// List of Strings.
FUNCTION_BLOCK FB_StringList
VAR
   List : ARRAY[0..GVL_List.LIST_SIZE - 1] OF T_MaxString; // hold list
   _Count : UDINT := 0; // number of items.
END_VAR

// Add item to list. TRUE if successful. 
METHOD PUBLIC AddItem : BOOL
VAR_INPUT
   Item : T_MaxString; // item to add.
END_VAR
IF _Count < GVL_List.LIST_SIZE THEN
   List[_Count] := Item; // list is zero indexed, so number of items points at next free space.
   _Count := _Count + 1;
   AddItem := TRUE;
END_IF
END_METHOD

// Removes all list items
METHOD PUBLIC Clear
MEMSET(ADR(List[0]), 0, SIZEOF(List));
_Count := 0;
END_METHOD

// TRUE if Item is in FB_List.
METHOD PUBLIC Contains : BOOL
VAR_INPUT
   Item : T_MaxString; // Item to check.
END_VAR
Contains := FindIndex(Item) >= 0;
END_METHOD

// TRUE if supplied key part is in any entry
METHOD PUBLIC ContainsPartial : BOOL
VAR_INPUT
   PartialItem : T_MaxString;
END_VAR
ContainsPartial := FindIndexPartialKey(PartialItem) >= 0;
END_METHOD

METHOD CopyList
VAR_IN_OUT
   ListToCopyTo : ARRAY[0..GVL_List.LIST_SIZE - 1] OF T_MaxString; // hold list
END_VAR
ListToCopyTo := THIS^.List;
END_METHOD

METHOD CopyListAndClear
VAR_IN_OUT
   ListToCopyTo : ARRAY[0..GVL_List.LIST_SIZE - 1] OF T_MaxString; // hold list
END_VAR
THIS^.CopyList(ListToCopyTo);
THIS^.Clear();
END_METHOD

{attribute 'monitoring' := 'call'}
// Number of items in list.
PROPERTY PUBLIC Count : UDINT
GET
Count := _Count;
END_GET
END_PROPERTY

METHOD PUBLIC FindIndex : INT
VAR_INPUT
   Item : T_MaxString; // Item to check.
END_VAR
VAR
   i : UINT := 0;
END_VAR
FindIndex := -1;
i := 0;

WHILE ((FindIndex < 0) AND (i < _Count)) DO

   FindIndex := SEL(Item = List[i], FindIndex, TO_INT(i)); // if it matches, return the position.
   i := i + 1;

END_WHILE
END_METHOD

// Find first index where list entry contains supplied key.
METHOD PUBLIC FindIndexPartialKey : INT
VAR_INPUT
   PartialKey : T_MaxString; // Item to check.
END_VAR
VAR
   i : UINT := 0;
END_VAR
FindIndexPartialKey := -1;
i := 0;

WHILE ((FindIndexPartialKey < 0) AND (i < _Count)) DO

   IF FIND(List[i], PartialKey) > 0 THEN
      FindIndexPartialKey := TO_INT(i);
   END_IF

   i := i + 1;

END_WHILE
END_METHOD

// Retrieve and remove the specified index.Failes silently
METHOD PUBLIC GetAndRemoveIndex : T_MaxString
VAR_INPUT
   Index : UDINT;
END_VAR
IF TryGetIndex(Index, GetAndRemoveIndex) THEN
   RemoveIndex(Index);
END_IF
END_METHOD

// Return item in list at index position. Returns empty string if invalid index.
METHOD PUBLIC GetIndex : T_MaxString
VAR_INPUT
   Index : UDINT;
END_VAR
THIS^.TryGetIndex(Index, GetIndex);
END_METHOD

//Remove the specified index. Shuffle remaining so list is intact.
METHOD PUBLIC RemoveIndex : BOOL
VAR_INPUT
   Index : UDINT;
END_VAR
IF Index >= _Count THEN // invalid index request.
   RETURN;
END_IF

IF Index < _Count - 1 THEN // If Index = _Count -1, last two lines sufficient.

   MEMMOVE(
      destAddr := ADR(List[Index]),
      srcAddr := ADR(List[Index + 1]),
      n := SIZEOF(List[0]) * (_Count - Index - 1)
   );

END_IF

RemoveIndex := TRUE;

List[_Count - 1] := ''; // default the "old" end of the list.
_Count := _Count - 1; // reduce count.
END_METHOD

// TRUE if successful and list item in sItem
METHOD PUBLIC TryGetIndex : BOOL
VAR_INPUT
   Index : UDINT;
END_VAR
VAR_IN_OUT
   Item : T_MaxString;
END_VAR
IF Index < _Count THEN
   TryGetIndex := TRUE;
   Item := List[Index];
END_IF
END_METHOD

END_FUNCTION_BLOCK

(* stored: Version 1.1.0.1, ProductVersion 3.1.4024.9
   POU FB_StringList: Id {5c73482d-8467-44b4-9630-4f585c9087e0}, SpecialFunc None
   Method AddItem: Id {51cf5f24-1e90-4b10-8307-a413650f5567}
   Method Clear: Id {bb59a1ae-0eeb-466d-95c9-57077c064997}
   Method Contains: Id {a309eed6-6ea3-4d92-8dd9-2037a6444569}
   Method ContainsPartial: Id {7a7f2235-0e70-49ce-ae3e-9202b3b1ec91}
   Method CopyList: Id {39a405c5-ca28-4471-b710-3b8972918780}
   Method CopyListAndClear: Id {c3e0a3e7-6839-4cd3-bbb6-f7d0188b7693}
   Property Count: Id {718e1bc0-d094-4e9e-81d3-a5637c94a50a}
   Get Get: Id {4590a6b8-077b-41b8-bc5b-3bb4b99253fe}
   Method FindIndex: Id {5adba4b6-ada1-4b43-b252-79c61e10ea0d}
   Method FindIndexPartialKey: Id {0617c0e9-f0f7-4092-8ade-c42aa34f7378}
   Method GetAndRemoveIndex: Id {d3dfb775-00be-4eca-b79a-9e227508aa2b}
   Method GetIndex: Id {fd53e871-2041-41d3-b12f-1eeb2e3044e7}
   Method RemoveIndex: Id {53807321-aeb2-4947-b125-ec03bf79b054}
   Method TryGetIndex: Id {22736251-d160-497b-8fff-8a6a25c6582d} *)
